// TIA Portal V20 export
TYPE "LKinCtrl_typeContourOffsetParameter"
   STRUCT
      "name" : String["LKINCTRL_LENGTH_OF_OFFSET_NAME"];   // offset name
      radius : LReal;   // offset radius
      length : LReal;   // offset length
   END_STRUCT;
END_TYPE
